FUNCTION_BLOCK Producer
  (* Standard: 61499-2 *)
  (* Version 0.1, 2017-00-09, hpea485, UOA *)
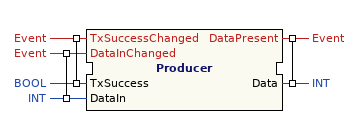
  EVENT_INPUT
    TxSuccessChanged WITH TxSuccess;
    DataInChanged WITH DataIn;
  END_EVENT
  EVENT_OUTPUT
    DataPresent WITH Data;
  END_EVENT
  VAR_INPUT
    TxSuccess : BOOL;
    DataIn : INT;
  END_VAR
  VAR_OUTPUT
    Data : INT;
  END_VAR
  VAR
    Count : INT := 0;
  END_VAR
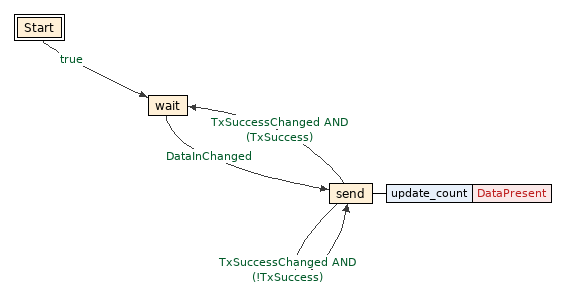
  EC_STATES
    Start;
    wait;
    send : update_count -> DataPresent;
  END_STATES
  EC_TRANSITIONS
    Start TO wait := true;
    wait TO send := DataInChanged;
    send TO wait := TxSuccessChanged AND (TxSuccess);
    send TO send := TxSuccessChanged AND (!TxSuccess);
  END_TRANSITIONS
  ALGORITHM update_count IN C:
me->Data = me->DataIn;
  END_ALGORITHM
END_FUNCTION_BLOCK
